// TIA Portal project "PLCII_Pro9" (V15.1)

(* hardware
DEVICE "S7-1200 station_1"  S7-1200 Station
   slot 0: "Rack_0"  S7-1200 Rack  Rack  V1.0
   slot 1: "PLC_1"  CPU 1215C DC/DC/Rly  6ES7 215-1HG40-0XB0  V4.2
DEVICE "HMI_1"  TP700 Comfort
   slot 0: "HMI_1"  TP700 Comfort  6AV2 124-0GC01-0AX0  15.1.0.0
   slot 1: "HMI_RT_1"  TP700 Comfort  6AV2 124-0GC01-0AX0  15.1.0.0
   slot 5: "HMI_1.IE_CP_1"  PROFINET Interface  15.0.1.0
      slot 1: "PROFINET Interface_1"  PROFINET Interface
         slot 1: "Port_1"  Port
         slot 2: "Port_2"  Port
   slot 7: "HMI_1.MPI/DP_CP_1"  MPI/DP Interface  15.0.1.0
*)

// ===== PLC "PLC_1"  CPU 1215C DC/DC/Rly =====

VAR_GLOBAL   // PLC tag table "Default tag table"
   "Start" AT %M0.0 : Bool;
   "Sys_runing" AT %M0.1 : Bool;
   "Stop" AT %M0.2 : Bool;
   "Activate" AT %M0.3 : Bool;
   "Sys_Activated" AT %M0.4 : Bool;
END_VAR

DATA_BLOCK "SysVaribales"   // DB1
{ S7_Optimized_Access := 'TRUE' }
VERSION : 0.1
   VAR
      SystemState : Int;
      CounterM1F1 : Int;
      CounterM1F2 : Int;
      CounterM2F1 : Int;
      CounterM2F2 : Int;
      CounterState : String;
   END_VAR
BEGIN
END_DATA_BLOCK

DATA_BLOCK "SystemCycles_DB"   // DB2
{ S7_Optimized_Access := 'TRUE' }
VERSION : 0.1
// stored: InstanceOfName SystemCycles
"SystemCycles"
BEGIN
END_DATA_BLOCK

DATA_BLOCK "TreateString_DB"   // DB3
{ S7_Optimized_Access := 'TRUE' }
VERSION : 0.1
// stored: InstanceOfName TreateString
"TreateString"
BEGIN
END_DATA_BLOCK

FUNCTION_BLOCK "SystemCycles"   // FB1, LAD
{ S7_Optimized_Access := 'TRUE' }
VERSION : 0.1
   VAR_INPUT
      Excute : Bool;
   END_VAR
   VAR
      ons1 : Bool;
      ons2 : Bool;
      ons3 : Bool;
      ons4 : Bool;
      ons5 : Bool;
      ons6 : Bool;
      ons7 : Bool;
      ons8 : Bool;
      ons9 : Bool;
      ons10 : Bool;
      ons11 : Bool;
      IEC_Timer_0_Instance : TON_TIME;
      IEC_Timer_0_Instance_1 : TON_TIME;
      IEC_Timer_0_Instance_2 : TON_TIME;
      IEC_Timer_0_Instance_3 : TON_TIME;
   END_VAR
   VAR CONSTANT
      Mode1 : Int := 1;
      Mode2 : Int := 2;
      Mode3 : Int := 3;
      Mode4 : Int := 4;
      TimeForFunction : Time := T#4s;
   END_VAR
   VAR_TEMP   // added for the SCL form of the ladder/FBD networks
      _w1 : Bool;
   END_VAR
BEGIN

REGION Network 1
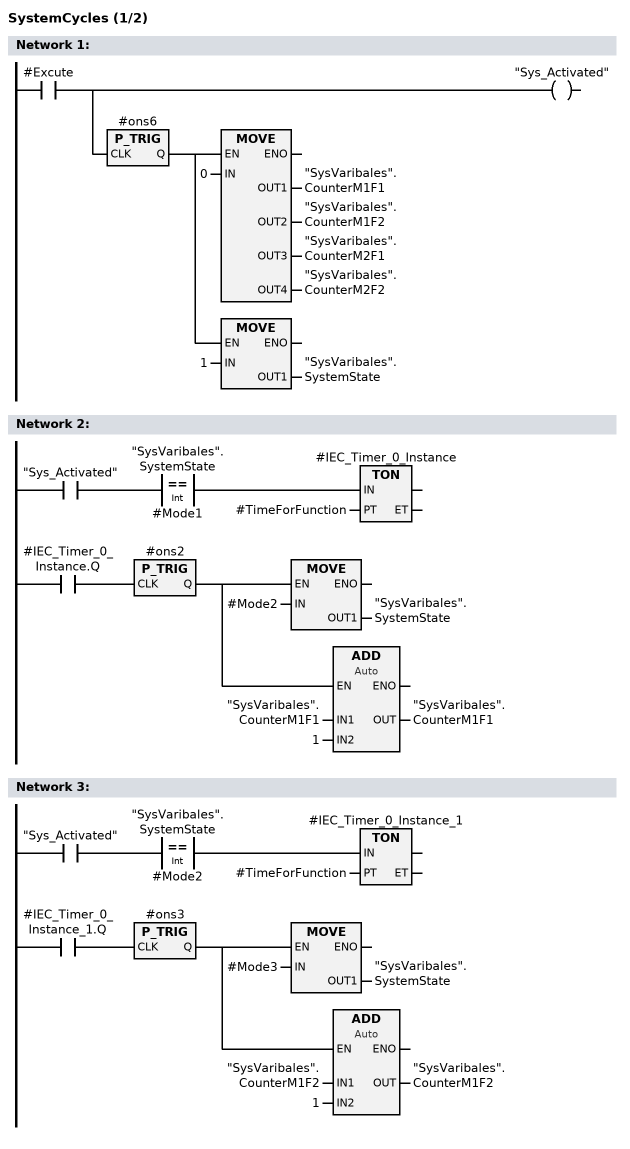
   RUNG wire#powerrail
      Contact( #Excute )
      wire#w1
      Coil( "Sys_Activated" )
   END_RUNG
   RUNG wire#w1
      P_Trig( #ons6 )
      wire#w2
      Move(in := 0, out1 => "SysVaribales".CounterM1F1, out2 => "SysVaribales".CounterM1F2, out3 => "SysVaribales".CounterM2F1, out4 => "SysVaribales".CounterM2F2)
   END_RUNG
   RUNG wire#w2
      Move(in := 1, out1 => "SysVaribales".SystemState)
   END_RUNG
   // the same network as SCL:
   "Sys_Activated" := #Excute;
   #_w1 := #Excute AND NOT #ons6;   // rising edge
   #ons6 := #Excute;
   IF #_w1 THEN
       "SysVaribales".CounterM1F1 := 0;
       "SysVaribales".CounterM1F2 := 0;
       "SysVaribales".CounterM2F1 := 0;
       "SysVaribales".CounterM2F2 := 0;
       "SysVaribales".SystemState := 1;
   END_IF;
END_REGION

REGION Network 2
   #IEC_Timer_0_Instance(IN := "Sys_Activated" AND ("SysVaribales".SystemState = #Mode1),   // TON
                         PT := #TimeForFunction);
   #_w1 := #IEC_Timer_0_Instance.Q AND NOT #ons2;   // rising edge
   #ons2 := #IEC_Timer_0_Instance.Q;
   IF #_w1 THEN
       "SysVaribales".SystemState := #Mode2;
       "SysVaribales".CounterM1F1 := "SysVaribales".CounterM1F1 + 1;
   END_IF;
END_REGION

REGION Network 3
   #IEC_Timer_0_Instance_1(IN := "Sys_Activated" AND ("SysVaribales".SystemState = #Mode2),   // TON
                           PT := #TimeForFunction);
   #_w1 := #IEC_Timer_0_Instance_1.Q AND NOT #ons3;   // rising edge
   #ons3 := #IEC_Timer_0_Instance_1.Q;
   IF #_w1 THEN
       "SysVaribales".SystemState := #Mode3;
       "SysVaribales".CounterM1F2 := "SysVaribales".CounterM1F2 + 1;
   END_IF;
END_REGION

REGION Network 4
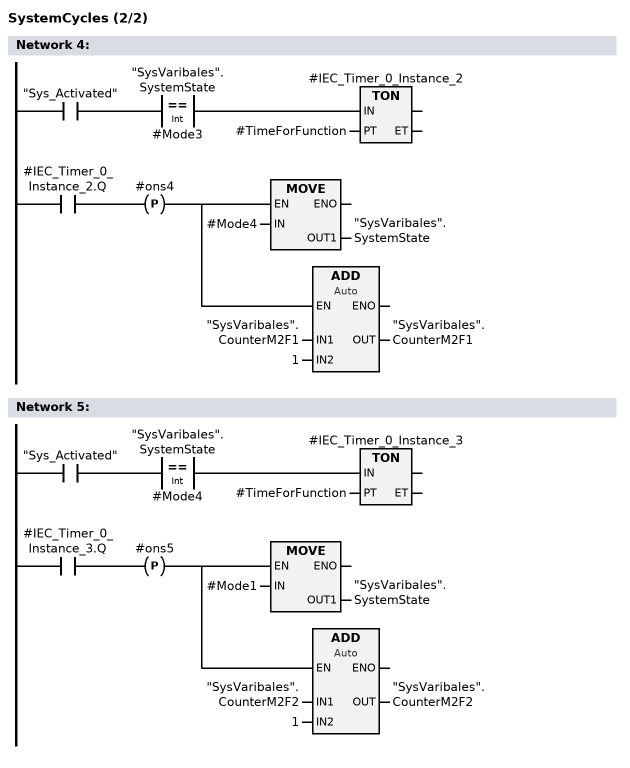
   #IEC_Timer_0_Instance_2(IN := "Sys_Activated" AND ("SysVaribales".SystemState = #Mode3),   // TON
                           PT := #TimeForFunction);
   #_w1 := #IEC_Timer_0_Instance_2.Q AND NOT #ons4;   // rising edge
   #ons4 := #IEC_Timer_0_Instance_2.Q;
   IF #_w1 THEN
       "SysVaribales".SystemState := #Mode4;
       "SysVaribales".CounterM2F1 := "SysVaribales".CounterM2F1 + 1;
   END_IF;
END_REGION

REGION Network 5
   #IEC_Timer_0_Instance_3(IN := "Sys_Activated" AND ("SysVaribales".SystemState = #Mode4),   // TON
                           PT := #TimeForFunction);
   #_w1 := #IEC_Timer_0_Instance_3.Q AND NOT #ons5;   // rising edge
   #ons5 := #IEC_Timer_0_Instance_3.Q;
   IF #_w1 THEN
       "SysVaribales".SystemState := #Mode1;
       "SysVaribales".CounterM2F2 := "SysVaribales".CounterM2F2 + 1;
   END_IF;
END_REGION
END_FUNCTION_BLOCK

FUNCTION_BLOCK "TreateString"   // FB2, LAD
{ S7_Optimized_Access := 'TRUE' }
VERSION : 0.1
   VAR_INPUT
      Excute : Bool;
   END_VAR
   VAR_OUTPUT
      StateOFFunctions : String;
   END_VAR
   VAR
      CM1F1 : String;
      CM1F2 : String;
      CM2F1 : String;
      CM2F2 : String;
   END_VAR
   VAR_TEMP
      StringTemp : String;
   END_VAR
   VAR CONSTANT
      ParaL : String := '(';
      ParaR : String := ')';
      Camma : String := ',';
   END_VAR
BEGIN

REGION Network 1
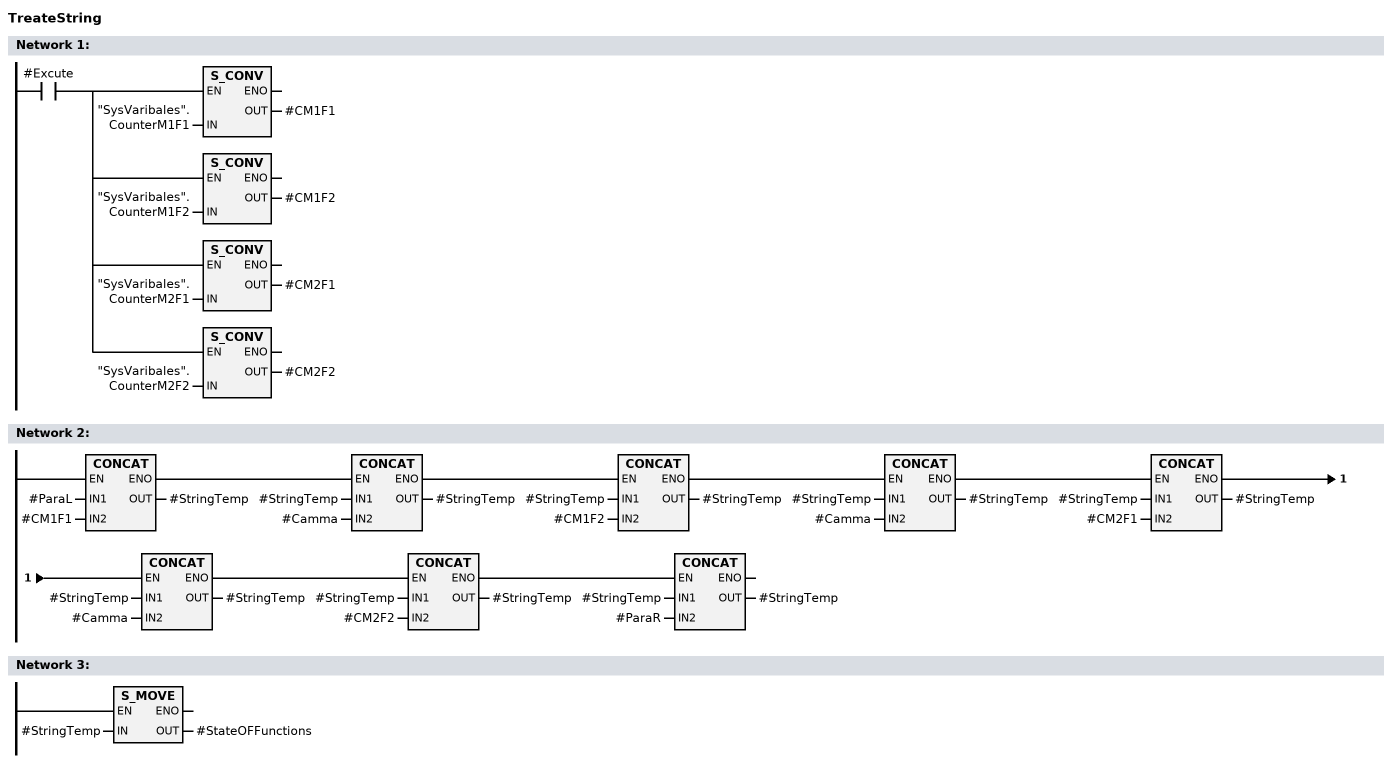
   IF #Excute THEN
       #CM1F1 := S_CONV(IN := "SysVaribales".CounterM1F1);
       #CM1F2 := S_CONV(IN := "SysVaribales".CounterM1F2);
       #CM2F1 := S_CONV(IN := "SysVaribales".CounterM2F1);
       #CM2F2 := S_CONV(IN := "SysVaribales".CounterM2F2);
   END_IF;
END_REGION

REGION Network 2
   #StringTemp := CONCAT(IN1 := #ParaL, IN2 := #CM1F1);
   #StringTemp := CONCAT(IN1 := #StringTemp, IN2 := #Camma);
   #StringTemp := CONCAT(IN1 := #StringTemp, IN2 := #CM1F2);
   #StringTemp := CONCAT(IN1 := #StringTemp, IN2 := #Camma);
   #StringTemp := CONCAT(IN1 := #StringTemp, IN2 := #CM2F1);
   #StringTemp := CONCAT(IN1 := #StringTemp, IN2 := #Camma);
   #StringTemp := CONCAT(IN1 := #StringTemp, IN2 := #CM2F2);
   #StringTemp := CONCAT(IN1 := #StringTemp, IN2 := #ParaR);
END_REGION

REGION Network 3
   RUNG wire#powerrail
      S_Move(in := #StringTemp, out => #StateOFFunctions)
   END_RUNG
   // the same network as SCL:
   #StateOFFunctions := #StringTemp;
END_REGION
END_FUNCTION_BLOCK

ORGANIZATION_BLOCK "Main"   // OB1, LAD, ProgramCycle
TITLE = "Main Program Sweep (Cycle)"
{ S7_Optimized_Access := 'TRUE' }
VERSION : 0.1
   VAR_INPUT
      Initial_Call : Bool;   // Initial call of this OB
      Remanence : Bool;   // =True, if remanent data are available
   END_VAR
BEGIN

REGION Network 1
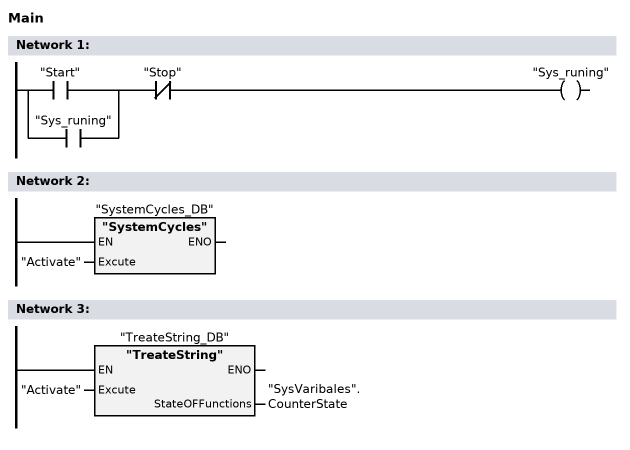
   RUNG wire#powerrail
      Contact( "Start" )
      wire#w1
      I_Contact( "Stop" )
      Coil( "Sys_runing" )
   END_RUNG
   RUNG wire#powerrail
      Contact( "Sys_runing" )
   END_RUNG wire#w1
   // the same network as SCL:
   "Sys_runing" := ("Start" OR "Sys_runing") AND NOT "Stop";
END_REGION

REGION Network 2
   RUNG wire#powerrail
      "SystemCycles_DB"(Excute := "Activate")
   END_RUNG
   // the same network as SCL:
   "SystemCycles_DB"(Excute := "Activate");   // "SystemCycles"
END_REGION

REGION Network 3
   RUNG wire#powerrail
      "TreateString_DB"(Excute := "Activate", StateOFFunctions => "SysVaribales".CounterState)
   END_RUNG
   // the same network as SCL:
   "TreateString_DB"(Excute := "Activate", StateOFFunctions => "SysVaribales".CounterState);   // "TreateString"
END_REGION
END_ORGANIZATION_BLOCK

(* ===== HMI "HMI_RT_1" =====
system functions are stored by id; their names below are inferred from use
connection "HMI_Connection_1": ETHERNET, S7_1200_OMS

HMI tags "Default tag table"
   "SysVaribales_CounterState" : String[254] = PLC SysVaribales.CounterState, 1 s
   "SysVaribales_SystemState" : Int = PLC SysVaribales.SystemState, 1 s

screen "Root screen" 800x420, template "Template_1"
   IOField "I/O field_1" at 70,46 size 501x32; FormatPattern ??????????????????????????????????????????????????????????????????????????????????????????????????????????????????????????????????????????????????????????????????????????????????????????????????????????????????????????????????????????????????????????????
      ProcessValue <- "SysVaribales_CounterState"
   IOField "I/O field_2" at 70,87 size 501x32; FormatPattern 99
      ProcessValue <- "SysVaribales_SystemState"
   Button "Button_1" at 210,130 size 222x32; TextOff 'ScriptTrigger'
      on Press: "VBFunction_1"()
      on Click: "VBFunction_1"()

Template "Template_1" 800x420
   Button "Exit" at 720,360 size 78x58; TextOff 'Exit'; PictureOff "ExitRuntime_TP700_Comfort_TR"; PictureOn "ExitRuntime_TP700_Comfort_TR"
      on Release: StopRuntime(0)
   Button "Template_Button" at 640,360 size 78x58; TextOff 'Text'
   Button "Template_Button_1" at 560,360 size 78x58; TextOff 'Text'
   Button "Template_Button_2" at 480,360 size 78x58; TextOff 'Text'
   Button "Template_Button_3" at 400,360 size 78x58; TextOff 'Text'
   Button "Template_Button_4" at 321,360 size 78x58; TextOff 'Text'
   Button "Template_Button_5" at 241,360 size 78x58; TextOff 'Text'
   Button "Template_Button_6" at 161,360 size 78x58; TextOff 'Text'
   Button "Alarms" at 81,360 size 78x58; TextOff 'Alarms'; PictureOff "AlarmDisplay_TP700_Comfort_TR"; PictureOn "AlarmDisplay_TP700_Comfort_TR"
      on Release: function_ef3f5d25("Alarm window_Unacknowledged", -1)
   Button "Start screen" at 1,360 size 78x58; TextOff 'Start screen'; PictureOff "NavigateHome_TP700_Comfort_TR"; PictureOn "NavigateHome_TP700_Comfort_TR"
      on Release: ActivateScreen("Root screen", 0)

VB script "VBFunction_1"
   'Tip:
   ' 1. Use the <CTRL+SPACE> or <CTRL+I> shortcut to open a list of all objects and functions
   ' 2. Write the code using the HMI Runtime object.
   '  Example: HmiRuntime.Screens("Screen_1").
   ' 3. Use the <CTRL+J> shortcut to create an object reference.
   'Write the code as of this position:
   ' Define Excel objects
   Dim objExcel, strExcelPath, strSaveAsPath, objSheet
   
   strExcelPath = "F:\file1.xlsx"
   strSaveAsPath = "F:\file1.xlsx"
   ' Open specified spreadsheet and select the first worksheet.
   Set objExcel = CreateObject("Excel.Application")
   objExcel.Workbooks.Open strExcelPath
   Set objSheet = objExcel.ActiveWorkbook.Worksheets(1)
   
   ' Write Cell value for the value.
   objSheet.Cells(2,2).Value = "0"
   objSheet.Cells(3,2).Value = SmartTags("SysVaribales_CounterState")
   
   ' Save and quit.
   'objExcel.ActiveWorkbook.Save
   objExcel.ActiveWorkbook.SaveAs strSaveAsPath
   objExcel.ActiveWorkbook.Close
   objExcel.Application.Quit
   
   ' SaveAs, Print and quit.
   
   objExcel.Workbooks.Open strSaveAsPath
   objExcel.ActiveWorkbook.PrintOut
   objExcel.ActiveWorkbook.Close
*)